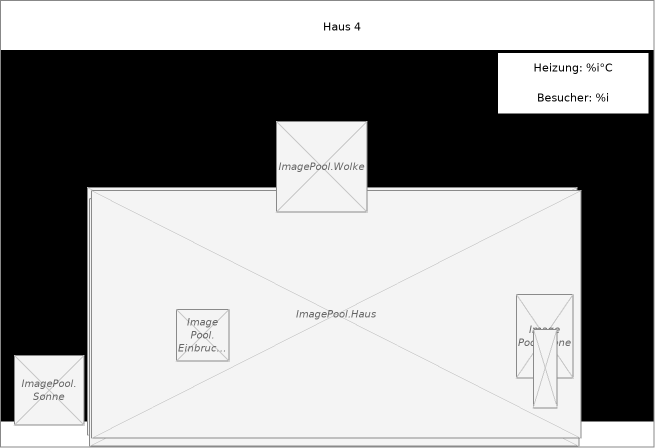
VISUALIZATION Haus_3  // 655x448
    Rectangle (1,50 652x371)
    Rectangle (1,50 652x371), colour variable: L_Himmel
        p2167032090: L_Himmel
    Image (87,187 490x248), invisible if: NOT net_licht_04, image: ImagePool.Dunkel
    Image (89,198 490x248), invisible if: net_licht_04, image: ImagePool.Licht
    Image (91,190 490x248), image: ImagePool.Haus
    Image (516,294 57x84), image: ImagePool.Krone
        p2858320360: L_Baum
    Image (533,329 24x79), image: ImagePool.Stamm
    Image (14,355 70x70), image: ImagePool.Sonne
        p2858320360: L_Sonnenstand
        p84334746: L_Sonne
    Image (176,309 53x52), image: ImagePool.Einbruch_grun
        p84334746: Haus4.L_EinbruchBild
    Image (276,121 91x91), image: ImagePool.Wolke
        p84334746: Haus4.WetterBild
    Textfield (267,16 150x22), "Haus 4"
    Textfield (498,53 150x30), "Heizung: %i°C", text variable: net_heizung_04
    Textfield (498,83 150x30), "Besucher: %i", text variable: net_besucher_04
END_VISUALIZATION

(* stored: Version 1.1.0.1, ProductVersion 3.1.4018.5
   Visu Haus_3: Id {7355bbbf-d0c4-42f4-91fa-77f3578973df} *)
